FUNCTION_BLOCK FB_UsingPiece EXTENDS FB_PieceBase
VAR_INPUT
END_VAR
VAR_OUTPUT
END_VAR
VAR
	bUsed 	: BOOL;	
END_VAR

METHOD M_GetAllProps : ERRORID
VAR_INPUT
	refCmdData : REFERENCE TO  ST_CmdData;
END_VAR
SUPER^.M_GetAllProps(refCmdData);
nCurrentPropIndex := nCurrentPropIndex + 1;
refCmdData.n32Data[nCurrentPropIndex] := BOOL_TO_DINT(bUsed);
END_METHOD

METHOD M_SetSingleProp : ERRORID
VAR_INPUT
	refCmdData : REFERENCE TO  ST_CmdData;
END_VAR
IF refCmdData.aHeader[1] = nSpecPropIndex THEN
	bUsed := DINT_TO_BOOL(refCmdData.n32Data[0]);
ELSE
	M_SetSingleProp := SUPER^.M_SetSingleProp(refCmdData);
END_IF
END_METHOD

{attribute 'object_name' := 'M_SetAllProps'}
METHOD M_SetAllProps : ERRORID
VAR_INPUT
	refCmdData	: REFERENCE TO ST_CmdData;
END_VAR
M_SetAllProps := SUPER^.M_SetAllProps(refCmdData);

IF M_SetAllProps > 0 THEN
	RETURN;
END_IF
nCurrentPropIndex := nCurrentPropIndex + 1;
nSpecPropIndex := nCurrentPropIndex;

bUsed := DINT_TO_BOOL(refCmdData.n32Data[nCurrentPropIndex]);

nNoOfProps := nCurrentPropIndex + 1;
END_METHOD

PROPERTY P_bUsed : BOOL
GET
P_bUsed := bUsed;
END_GET
SET
bUsed := P_bUsed;
END_SET
END_PROPERTY

END_FUNCTION_BLOCK

(* stored: Version 1.1.0.1, ProductVersion 3.1.4020.12
   POU FB_UsingPiece: Id {589d7b24-c269-4556-930d-758c14b4d4bd}, SpecialFunc None
   Method M_GetAllProps: Id {00896a53-b4b1-4de5-aaab-a48bd8ebf8ab}
   Method M_SetSingleProp: Id {09b234f1-46ac-4429-88b5-2ded79f947a0}
   Method M_SetAllProps: Id {a31952c0-cdcd-490c-9d67-9c629746b449}
   Property P_bUsed: Id {f4e29365-f381-4d88-bf7f-4e2a0d584453}
   Get Get: Id {9ef46ae1-fbda-4e3b-a20b-93656b63742c}
   Set Set: Id {e1899119-3c06-4289-afcf-8aae6feedf15} *)
